FUNCTION_BLOCK INTERNAL FB_MotionLogger_Test EXTENDS FB_TestSuite

VAR

END_VAR

GetLastWarningMessage_Test1();

METHOD PRIVATE GetLastWarningMessage_Test1
VAR_INST
	logs : STRING(1024);
	fbMotionLogger : FB_MotionLogger ;
END_VAR
TEST(__POUNAME());
fbMotionLogger.Clear();
fbMotionLogger.Logger(Message := 'One', Level := E_MotionLogLevel.INFO, Source := 'A');
fbMotionLogger.Logger(Message := 'Two', Level := E_MotionLogLevel.WARNING, Source := 'B');
fbMotionLogger.Logger(Message := 'Three', Level := E_MotionLogLevel.ERROR, Source := 'C');

logs := fbMotionLogger.GetAllMessages();

AssertTrue(
    Condition := FIND(logs, 'One') > 0 AND FIND(logs, 'Two') > 0 AND FIND(logs, 'Three') > 0,
    Message := 'GetAllMessages should include all log entries'
);
fbMotionLogger.Clear();

AssertTrue(
    Condition := fbMotionLogger.GetMessageCount() = 0,
    Message := 'Logger buffer must be empty'
);

TEST_FINISHED();
END_METHOD

END_FUNCTION_BLOCK

(* stored: Version 1.1.0.1
   POU FB_MotionLogger_Test: Id {d95d87fd-299b-4a22-9f20-cceebae3e038}, SpecialFunc None
   Method GetLastWarningMessage_Test1: Id {86c45580-5f09-4e83-a7a3-2f36de9a4ff9} *)
